FUNCTION_BLOCK ADD_WITH_SCALAR_FACTOR (* Setups data for main slot loop *)
  (* Standard: 61499-2 *)
  (* Version 1.0, 25-05-12, GASR, Universidade do Estado de Santa Catarina *)
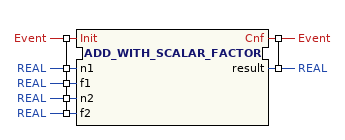
  EVENT_INPUT
    Init WITH n1, f1, n2, f2;
  END_EVENT
  EVENT_OUTPUT
    Cnf WITH result;
  END_EVENT
  VAR_INPUT
    n1 : REAL;
    f1 : REAL; (* f multiplies n *)
    n2 : REAL;
    f2 : REAL; (* f multiplies n *)
  END_VAR
  VAR_OUTPUT
    result : REAL;
  END_VAR
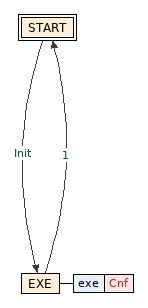
  EC_STATES
    START;
    EXE : exe -> Cnf;
  END_STATES
  EC_TRANSITIONS
    START TO EXE := Init;
    EXE TO START := 1;
  END_TRANSITIONS
  ALGORITHM exe IN Lua:
result = f1*n1 + f2*n2
print( result, f1, n1, f2, n2 )
  END_ALGORITHM
END_FUNCTION_BLOCK
